# EPICS autosave request: iocBoot/iocagilent33521a/auto_settings_EgunTest.req
file "agilent33521_EgunTest.req",                P=$(P),  R=$(R)
